(* PLC project v0.6.02_RefactorGateAndTest.project, CODESYS CODESYS V3.5 SP19 Patch 1 *)
(* stored: creationDateTime 2026-08-16T00:42:51.247269, modificationDateTime 2026-08-16T00:42:51.247269 *)

(* ═══════════════════════════════════════════════════════════════ 💾 PRG_Pool — Traitement des jobs async CAA File ─────────────────────────────────────────────────────────────── 🎯 Rôle : appelle le pool extender chaque cycle (dans la tâche 'myPoolExtender') pour traiter les jobs async d'écriture fichier. 📄 Docs : bibliothèque RSU + CAA File. ═══════════════════════════════════════════════════════════════ *)
PROGRAM PRG_Pool

            GVL_Pool.myPoolExtender;   // traite les jobs async chaque cycle

          
END_PROGRAM
